// Mitsubishi GX Works2 project: De10   PLC: FX2N/FX2NC

PROGRAM MAIN
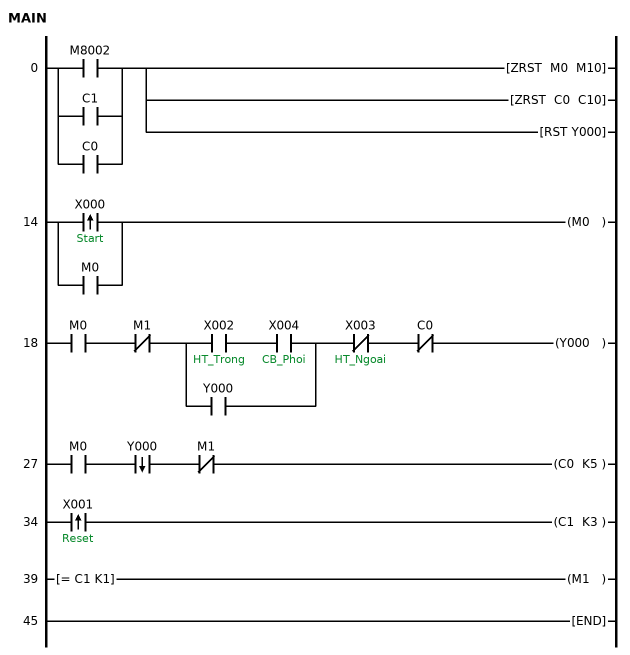
0     LD      M8002
      OR      C1
      OR      C0
      ZRST    M0 M10
      ZRST    C0 C10
      RST     Y000
14    LDP     X000  ; Start
      OR      M0
      OUT     M0
18    LD      M0
      ANI     M1
      LD      X002  ; HT_Trong
      AND     X004  ; CB_Phoi
      OR      Y000
      ANB
      ANI     X003  ; HT_Ngoai
      ANI     C0
      OUT     Y000
27    LD      M0
      ANDF    Y000
      ANI     M1
      OUT     C0 K5
34    LDP     X001  ; Reset
      OUT     C1 K3
39    LD=     C1 K1
      OUT     M1
45    END
END_PROGRAM
